(* Logix 5000 project; controller PLCbox vendor 1 type 14 code 149 rev 30.11; software revision 30.01; part 3 of 3 *)
(* TestProgram, continued *)

ROUTINE Main   (* ladder *)
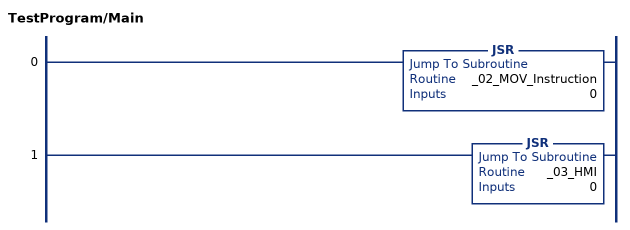
   0: JSR(_02_MOV_Instruction,0);
   1: JSR(_03_HMI,0);
END_ROUTINE
END_PROGRAM
